FUNCTION_BLOCK ContentFilter (* FB to check if a member value is changed or no! *)
  (* Standard: 61499-2 *)
  (* Version 1.0, 2021-07-23, AK121668 *)
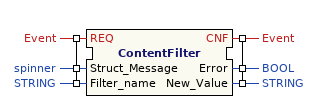
  EVENT_INPUT
    REQ WITH Filter_name, Struct_Message;
  END_EVENT
  EVENT_OUTPUT
    CNF WITH Error, New_Value;
  END_EVENT
  VAR_INPUT
    Struct_Message : spinner;
    Filter_name : STRING;
  END_VAR
  VAR_OUTPUT
    Error : BOOL;
    New_Value : STRING;
  END_VAR
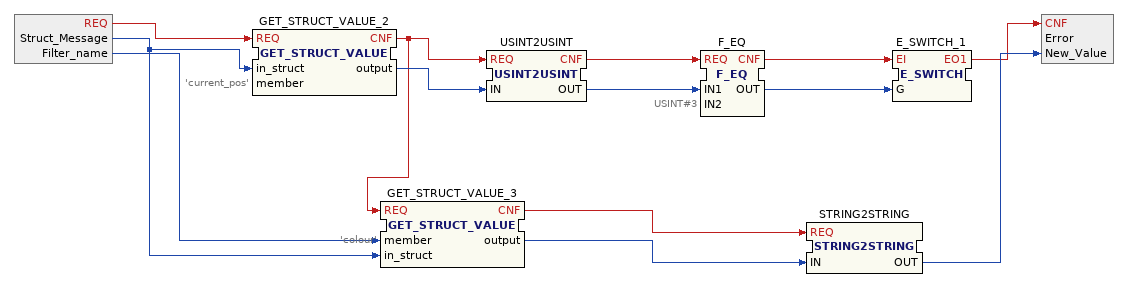
  FBS
    GET_STRUCT_VALUE_2 : GET_STRUCT_VALUE(member := 'current_pos');
    E_SWITCH_1 : E_SWITCH;
    GET_STRUCT_VALUE_3 : GET_STRUCT_VALUE(member := 'colour');
    STRING2STRING : STRING2STRING;
    F_EQ : F_EQ(IN2 := USINT#3);
    USINT2USINT : USINT2USINT;
  END_FBS
  EVENT_CONNECTIONS
    F_EQ.CNF TO E_SWITCH_1.EI;
    GET_STRUCT_VALUE_3.CNF TO STRING2STRING.REQ;
    GET_STRUCT_VALUE_2.CNF TO GET_STRUCT_VALUE_3.REQ;
    E_SWITCH_1.EO1 TO CNF;
    REQ TO GET_STRUCT_VALUE_2.REQ;
    USINT2USINT.CNF TO F_EQ.REQ;
    GET_STRUCT_VALUE_2.CNF TO USINT2USINT.REQ;
  END_CONNECTIONS
  DATA_CONNECTIONS
    GET_STRUCT_VALUE_3.output TO STRING2STRING.IN;
    F_EQ.OUT TO E_SWITCH_1.G;
    STRING2STRING.OUT TO New_Value;
    Filter_name TO GET_STRUCT_VALUE_3.member;
    USINT2USINT.OUT TO F_EQ.IN1;
    GET_STRUCT_VALUE_2.output TO USINT2USINT.IN;
    Struct_Message TO GET_STRUCT_VALUE_2.in_struct;
    Struct_Message TO GET_STRUCT_VALUE_3.in_struct;
  END_CONNECTIONS
END_FUNCTION_BLOCK
